INTERFACE I_DS402PiezoDrive

METHOD Brake
VAR_INPUT
END_VAR
END_METHOD

METHOD EncSaveRestore
VAR_INPUT
	 bEnable: BOOL;
END_VAR
END_METHOD

METHOD EncValue
VAR_INPUT
//    bEnable: BOOL;
END_VAR
END_METHOD

{attribute 'monitoring':= 'variable'}
PROPERTY Error : BOOL
GET
END_GET
SET
END_SET
END_PROPERTY

{attribute 'monitoring':= 'variable'}
PROPERTY ErrorCode : UDINT
GET
END_GET
SET
END_SET
END_PROPERTY

{attribute 'monitoring':= 'variable'}
PROPERTY ErrorMessage : STRING
GET
END_GET
SET
END_SET
END_PROPERTY

METHOD Halt : BOOL
VAR_INPUT
END_VAR
END_METHOD

METHOD Home : BOOL
VAR_INPUT
END_VAR
END_METHOD

{attribute 'monitoring':= 'variable'}
PROPERTY HomeDone : BOOL
GET
END_GET
SET
END_SET
END_PROPERTY

{attribute 'monitoring':= 'variable'}
PROPERTY HomingBusy : BOOL
GET
END_GET
SET
END_SET
END_PROPERTY

METHOD Interlock
VAR_INPUT
END_VAR
END_METHOD

METHOD Logger
VAR_INPUT
END_VAR
END_METHOD

METHOD MotionParams
VAR_INPUT
    tRefreshDelay: TIME;
END_VAR
END_METHOD

METHOD MoveAbsolute
VAR_INPUT
END_VAR
END_METHOD

{attribute 'monitoring':= 'variable'}
PROPERTY MoveBusy : BOOL
GET
END_GET
SET
END_SET
END_PROPERTY

{attribute 'monitoring':= 'variable'}
PROPERTY MoveDone : BOOL
GET
END_GET
SET
END_SET
END_PROPERTY

METHOD MoveVelocity
VAR_INPUT
END_VAR
END_METHOD

METHOD Power : BOOL
VAR_INPUT
END_VAR
END_METHOD

METHOD Reset : BOOL
VAR_INPUT
END_VAR
END_METHOD

METHOD SetEnables
VAR_INPUT
END_VAR
END_METHOD

METHOD StateMachine
VAR_INPUT
END_VAR
END_METHOD

END_INTERFACE

(* stored: Version 1.1.0.1
   Itf I_DS402PiezoDrive: Id {49729736-8717-4a13-800f-a53162ccda84}
   Method Brake: Id {e0529470-e1a2-408b-acaa-cacbe414aa6e}
   Method EncSaveRestore: Id {2714254e-be9f-442a-9ff0-fec0cfde8ef7}
   Method EncValue: Id {5a3e0ac7-04c3-493b-9cb6-07a60972201e}
   Property Error: Id {ecddf92f-389a-4b66-a847-9288fadbdd07}
   Get Get: Id {3995c37e-c525-4213-a810-2df3fd6c72d0}
   Set Set: Id {787eda39-89c4-4a82-b023-e351d7cb86c7}
   Property ErrorCode: Id {83ccf468-2f12-4981-a5ae-5955a7f86878}
   Get Get: Id {83114e97-87ef-4199-9ca8-05ef0c812ee8}
   Set Set: Id {86d20c2b-16b5-44f9-b245-31a20d41dde9}
   Property ErrorMessage: Id {5b6e842b-7143-43fe-83dd-a3d6fb4ab9ed}
   Get Get: Id {1c19bdcc-bf5e-4bbf-af14-21e46885d40d}
   Set Set: Id {fc52c698-0a25-4b7c-a6f2-167c5ce1faf7}
   Method Halt: Id {1645d0ef-eb4b-4235-b6cc-4a214463d443}
   Method Home: Id {f7b9941e-fd39-45a3-99c7-fc867c3625ba}
   Property HomeDone: Id {200cd3be-65e8-40a3-9d86-5f57e4e0faf5}
   Get Get: Id {b1028f7c-ce5a-4deb-bc48-6a75b8249228}
   Set Set: Id {8c6b0f72-0c3a-491e-8005-de763463ac1c}
   Property HomingBusy: Id {ccf273c0-b5d1-46d7-89a2-f64672010979}
   Get Get: Id {4350797f-1e59-4083-b7c2-86586cc287ad}
   Set Set: Id {4aa1be67-b2f0-46e0-aecb-85c18cbef79b}
   Method Interlock: Id {b9614087-83f0-4675-8dad-b6765017e9ea}
   Method Logger: Id {36d29a03-8107-42f2-b596-87523b11c29f}
   Method MotionParams: Id {26e38a32-22d0-42ae-b0c6-5a30c1359c2c}
   Method MoveAbsolute: Id {c32a9e13-f332-4841-9fc3-9751e2083446}
   Property MoveBusy: Id {d0e70aa3-dd5f-4993-80bc-c333f23353c3}
   Get Get: Id {2ff17fdf-37b3-4f53-933b-aa2caf936d99}
   Set Set: Id {b7604329-d89a-4af5-b773-b6e19b1e5f38}
   Property MoveDone: Id {90606f0a-a16a-4ffe-93ef-405ecad06807}
   Get Get: Id {0ae3f37d-a00f-4d46-89b6-82fdb536fd4e}
   Set Set: Id {d0d57c30-381a-47aa-a3c5-49b7443da0de}
   Method MoveVelocity: Id {bc7db01d-6c11-4d35-a626-79d63771cf0a}
   Method Power: Id {08548eb9-8f7d-4758-8069-c44e4c6df0ba}
   Method Reset: Id {43fc3192-2758-4d04-872e-08906cd5bf28}
   Method SetEnables: Id {b93a945e-5ba8-456d-9ebc-47294f36ee3e}
   Method StateMachine: Id {35531d1d-083e-4e0e-a309-4f04090b40cb} *)
